// Mitsubishi GX Works2 project: ZhaoQing_ChengPinKu_Debug   PLC: Q03UDE
// 化成线2号柜

TYPE BarCylinderIO : STRUCT
  xPresentSwitch : BOOL;  (* 行程开关 *)
  xBarCylinder : BOOL;  (* 阻挡气缸 *)
  xEmpty : BOOL;  (* 为空指示 *)
  xTransportMotorCW : BOOL;  (* 输送电机正转 *)
  tLeaveDelay : TIME;  (* 放行延时 *)
  xUnload : BOOL;  (* 下料 *)
  xBarCylinderButton : BOOL;  (* 阻挡气缸 *)
  xTransportMotorCWButton : BOOL;  (* 输送电机正转按钮 *)
  xLoad : BOOL;  (* 上料 *)
  xNextRun : BOOL;  (* 下位设备开始运行 *)
  xTransportMotorCCWButton : BOOL;  (* 输送电机反转按钮 *)
  xTransportMotorCCW : BOOL;  (* 输送电机反转 *)
END_STRUCT END_TYPE

TYPE ConveyorIO : STRUCT
  xCWPresent : BOOL;  (* 正转检测有无传感器 *)
  xCCWPresent : BOOL;  (* 反转检测有无传感器 *)
  xLoad : BOOL;  (* 上料请求 *)
  xUnload : BOOL;  (* 下料请求 *)
  xMotorCW : BOOL;  (* 电机正转 *)
  xMotorCCW : BOOL;  (* 电机反转 *)
  xEmpty : BOOL;  (* 线体状态为空 *)
  xNextRun : BOOL;  (* 下段线体运行 *)
  xUnloadCCW : BOOL;  (* 下料为反转 *)
  xloadCCW : BOOL;  (* 上料为反转 *)
  xLeave : BOOL;  (* 已经离开 *)
  xForward : BOOL;  (* 正转手动 *)
  xBackward : BOOL;  (* 反转手动 *)
  xBusy : BOOL;  (* 工作中 *)
  xPutInto : BOOL;  (* 线体直接投入物料 *)
  xUnloadAlarm : BOOL;  (* 下料报警 *)
  tLoadDelay : TIME;  (* 进入延时设置 *)
  xPosLimit : BOOL;  (* 正限位 *)
  xNegLimit : BOOL;  (* 负限位 *)
  xOverWidthAlarm : BOOL;  (* 超宽报警 *)
  xLimitAlarrm : BOOL;  (* 限位报警 *)
  iDeviceID : INT;  (* 线体ID *)
END_STRUCT END_TYPE

TYPE RGVCommunication : STRUCT
  xFullLoadRequest : BOOL;  (* 满框上料请求 *)
  xFullUnloadRequest : BOOL;  (* 满框下料请求 *)
  xEmptyLoadRequest : BOOL;  (* 空框上料请求 *)
  xEmptyUnloadRequest : BOOL;  (* 空框下料请求 *)
  xFullLoadRequestAkn : BOOL;  (* 满框上料请求确认 *)
  xFullUnloadRequestAkn : BOOL;  (* 满框下料请求确认 *)
  xEmptyLoadRequestAkn : BOOL;  (* 空框上料请求确认 *)
  xEmptyUnloadRequestAkn : BOOL;  (* 空框下料请求确认 *)
  xFullLoadComplete : BOOL;  (* 满框上料完成 *)
  xFullUnloadComplete : BOOL;  (* 满框下料完成 *)
  xEmptyLoadComplete : BOOL;  (* 空框上料完成 *)
  xEmptyUnloadComplete : BOOL;  (* 空框下料完成 *)
  xFullLoadCompleteAkn : BOOL;  (* 满框上料完成确认 *)
  xFullUnloadCompleteAkn : BOOL;  (* 满框下料完成确认 *)
  xEmptyLoadCompleteAkn : BOOL;  (* 空框上料完成确认 *)
  xEmptyUnloadCompleteAkn : BOOL;  (* 空框下料完成确认 *)
END_STRUCT END_TYPE

TYPE ShuttleCarIO : STRUCT
  xReady : BOOL;  (* 准备就绪 *)
  xForward : BOOL;  (* 正转 *)
  xBackward : BOOL;  (* 反转 *)
  iCurrentPos : INT;  (* 当前位置 *)
  iDestinationPos : INT;  (* 目标位置 *)
  xCW : BOOL;  (* 正转输出 *)
  xCCW : BOOL;  (* 反转输出 *)
  xBrake : BOOL;  (* 刹车 *)
  xHomeSwitch : BOOL;  (* 零位接近开关 *)
  xPosLimit : BOOL;  (* 正限位 *)
  xNegLimit : BOOL;  (* 负限位 *)
  xMDIExe : BOOL;  (* MDI开始 *)
  xMDIDone : BOOL;  (* MDI 完成 *)
  xPassLimit : BOOL;  (* 限位屏蔽 *)
  xPosLimitCatch : BOOL;  (* 正限位捕捉 *)
  xNegLimitCatch : BOOL;  (* 负限位捕捉 *)
  xHomeExe : BOOL;  (* 开始寻零 *)
  xHomeDone : BOOL;  (* 寻零完成 *)
  xHomeBusy : BOOL;  (* 寻零中 *)
  xHomeFailed : BOOL;  (* 寻零失败 *)
  xBusy : BOOL;  (* 工作中 *)
  tArriveDelay : TIME;  (* 到位延时 *)
  xCylinder : BOOL;  (* 气缸控制 *)
  tBrakeDelay : TIME;  (* 抱闸延时 *)
  xPauseRamp : BOOL;  (* 暂停减速斜坡标志位 *)
  xPresentDetect1 : BOOL;  (* 物料有无检测1 *)
  xPresentDetect2 : BOOL;  (* 物料有无检测2 *)
  xOvertimeAlarm : BOOL;  (* 超时报警 *)
  tSetOverTime : TIME;  (* 设置超时时间 *)
  xLooseDetect : BOOL;  (* 松绳检测 *)
  xLooseAlarm : BOOL;  (* 松绳报警 *)
END_STRUCT END_TYPE

TYPE SwitchIO : STRUCT
  xLiftCylinderRetractDetect : BOOL;
  xLiftCylinderExtendDetect : BOOL;
  xLiftCylinderRetract : BOOL;
  xLiftCylinderExtend : BOOL;
  xEntryBarCylinderRetract : BOOL;
  xExitBarCylinderRetract : BOOL;
  xLiftCylinderExtendInit : BOOL;
  xEntryEnable : BOOL;
  xExitEnable : BOOL;
  xSwithEnable : BOOL;
  xLiftCylinderRetractButton : BOOL;
  xLiftCylinderExtendButton : BOOL;
  xEntryBarCylinderRetractButton : BOOL;
  xExitBarCylinderRetractButton : BOOL;
  xPutInto : BOOL;  (* 单体复位 *)
  tSetOvertime : TIME;  (* 设定超时报警时间 *)
  xOvertimeAlarm : BOOL;  (* 超时报警 *)
END_STRUCT END_TYPE

// global labels: Global1
VAR_GLOBAL
  g_xAuto AT M11 : BOOL;  (* 自动 *)
  g_xManual : BOOL;  (* 手动 *)
  g_xEStop : BOOL;  (* 急停 *)
  g_xReset : BOOL;  (* 复位 *)
  g_xStackLampRed : BOOL;
  g_xStackLampAmber : BOOL;
  g_xStackLampGreen : BOOL;
  g_xBuzzer : BOOL;
  g_xStop AT M2 : BOOL;  (* 停止 *)
  g_xLocalAutoStart AT M1 : BOOL;
  g_xRemoteAutoStart AT M0 : BOOL;
  g_xRemoteAuto AT M10 : BOOL;
  g_iState AT D40 : INT;
  g_iLocalAutoStep : INT;
  g_xError : BOOL;
  g_xStart : BOOL;  (* 启动 *)
  g_xResetSingle AT M4 : BOOL;  (* 单线体复位 *)
  g_iDeviceIDSelect AT D0 : INT;
  g_xPause AT M3 : BOOL;  (* 暂停 *)
END_VAR

// task Task_01 (event TRUE, interval 0, priority 31): Start, POU

FUNCTION_BLOCK BarCylinder
VAR_IN_OUT
  BarCylinderIO : BarCylinderIO;
END_VAR
VAR
  m_tonViaDelay : TON;  (* 卸料延时定时器 *)
  m_xViaDelay : BOOL;  (* 通过延时 *)
  m_tViaDelayElapse : TIME;  (* 通过延时当前时间 *)
  m_xInitial : BOOL;  (* 初始化 *)
END_VAR
  (***********************************************************************
阻挡器模块，
由一个行程开关，一个阻挡器，一个倍速链输送电机组成
具有手动与自动模式
xEmpty显示当前为空料的状态
xUnload为卸料信号，连接下一设备的xEmpty信号
*************************************************************************)

  (*初始化，离开延时时间设置为5秒*)
IF NOT m_xInitial THEN
	 BarCylinderIO.tLeaveDelay :=T#5s;
	m_xInitial:=1;
END_IF;
IF g_xManual THEN    (*手动*)
	BarCylinderIO.xNextRun:=0;
	IF BarCylinderIO.xBarCylinderButton THEN
		BarCylinderIO.xBarCylinder:=1;
	ELSE
		BarCylinderIO.xBarCylinder:=0;
	END_IF;
	IF BarCylinderIO.xTransportMotorCWButton 
		AND NOT BarCylinderIO.xTransportMotorCCWButton 
		AND NOT BarCylinderIO.xTransportMotorCCW   THEN
		BarCylinderIO.xTransportMotorCW:=1;
	ELSE
		BarCylinderIO.xTransportMotorCW:=0;
	END_IF;
	IF BarCylinderIO.xTransportMotorCCWButton 
		AND NOT BarCylinderIO.xTransportMotorCWButton 
		AND NOT BarCylinderIO.xTransportMotorCW   THEN
		BarCylinderIO.xTransportMotorCCW:=1;
	ELSE
		BarCylinderIO.xTransportMotorCCW:=0;
	END_IF;
END_IF;
(*离开延时定时器*)
m_tonViaDelay(IN:=NOT  BarCylinderIO.xPresentSwitch AND g_xAuto  ,PT:= BarCylinderIO.tLeaveDelay ,Q:= BarCylinderIO.xEmpty ,ET:=m_tViaDelayElapse );

IF g_xAuto THEN(*自动*)
    IF BarCylinderIO.xUnload  AND NOT BarCylinderIO.xEmpty AND NOT BarCylinderIO.xNextRun THEN(*收到卸料命令，当阻挡器不为空时*)
    	BarCylinderIO.xBarCylinder:=1;
    	BarCylinderIO.xNextRun:=1;(*确保下料命令只执行一次，防止物料在输送过程中又有卸料命令导致多事卸料*)
    	BarCylinderIO.xTransportMotorCW:=1;
    END_IF;
    IF NOT  BarCylinderIO.xUnload  THEN
    	BarCylinderIO.xNextRun:=0;
    END_IF;
    (*如果为空，气缸顶起*)
   IF  BarCylinderIO.xEmpty  THEN
   	   BarCylinderIO.xBarCylinder:=0;
   	   IF BarCylinderIO.xLoad THEN
	   	   BarCylinderIO.xTransportMotorCW:=1;
	   END_IF;
   END_IF;
   IF NOT BarCylinderIO.xUnload AND NOT  BarCylinderIO.xEmpty THEN
   	    BarCylinderIO.xTransportMotorCW:=0;
   	END_IF;
END_IF;
IF NOT g_xEStop THEN
	 BarCylinderIO.xTransportMotorCW:=0;
	 BarCylinderIO.xTransportMotorCCW:=0;
	 BarCylinderIO.xBarCylinder:=0;
END_IF;
END_FUNCTION_BLOCK

FUNCTION_BLOCK Conveyor
VAR
  tRundelay : TIME;  (* 离开延时 *)
END_VAR
VAR_IN_OUT
  ConveyorMotor : ConveyorIO;  (* 输送线输入输出 *)
END_VAR
VAR
  iStep : INT;  (* 上料步骤 *)
  m_tUnloadTimer : TIME;  (* 下料计时器 *)
  m_tonLeaveDelay : TON;  (* 离开延时定时器 *)
  m_xLeaveDelayOut : BOOL;  (* 离开延时 *)
  m_tLeaveCurrentTime : TIME;
END_VAR
VAR CONSTANT
  LOAD_UNLOAD_TIME : TIME := T#30s;  (* 延时报警常量 *)
END_VAR
VAR
  m_tonUnloadAlam : TON;  (* 下料报警定时器 *)
  m_tonLoadDelay : TON;  (* 离开延时定时器 *)
  m_xLoadDelayOut : BOOL;  (* 离开延时 *)
  m_tLoadCurrentTime : TIME;
  m_xInitial : BOOL;  (* 初始化 *)
  m_tLoadTimer : TIME;  (* 上料延时当前时间 *)
END_VAR
(*////////////////////////////////////////////////////////////////////////////////////////////////////////////
//传输线控制FB块，可控制单方向线体，双向旋转线体，支持双向上下料            
//线体初始化后为空的情况下输入xLoad信号即可进行上料动作，使用xLoadCCW信号可反方向上料
//增加了产品信息和产品种类的储存，当传输线为空和上料进行标志位为零的情况下清除产品信息和产品种类
//使用方式是在置位xLoad信号后，把产品信息和产品种类传入，等下料后自动清零
//线体不为空的情况下使用xUnload信号可进行下料动作，物料有无传感器的下降沿后出发计时器，延时断开传输线旋转
//单方向传输线体把xLoadCCW、xUnloadCCW设置为零，双向线体上料方向和下料反向的,方向固定的 把xUnloadCCW设置为1
//双方向线体双向都能上下料的要根据上料的方向来设置xLoadCCW,xUnloadCCW
//增加工作中信号xBusy当电机正转 显示为工作中
//增加上下料超时报警，xLoadAlarm，xUnloadAlarm，设定时间在LOAD_UNLOAD_TIME常量上，现在设置的为30秒
//增加xPutInto信号，用于直接投入的物料，检测开关感应到后，直接进入下料流程，上升沿有效
//离开延时改为变量 iLeaveDelay 默认为0 离开检测开关离输送线尾端比较远的线体需要根据情况设定100ms为单位
增加初始化标志位，增加进入延时时间，初始化为进入延时时间为0 ，离开延时时间为2S，通过外围接口可以更改
//修改信息  修改后请增加版本
//YAO      V1.0
///////////////////////////////////////////////////////////////////////////////////////////////////////////
********************************************************)
IF NOT m_xInitial THEN
	ConveyorMotor.tLoadDelay:=T#100ms;
	ConveyorMotor.xNegLimit:=1;
	ConveyorMotor.xPosLimit:=1;
END_IF;
m_xInitial:=1;
IF g_xAuto THEN
CASE iStep OF
	0:
	ConveyorMotor.xMotorCW:=0;
	ConveyorMotor.xMotorCCW:=0;
	ConveyorMotor.xNextRun:=0;
IF g_xEStop AND NOT ConveyorMotor.xLimitAlarrm  THEN
	IF (ConveyorMotor.xCWPresent OR ConveyorMotor.xCCWPresent)  THEN
		iStep:=3;
		ConveyorMotor.xEmpty:=0;
		ELSE
		iStep:=1;
		ConveyorMotor.xEmpty:=1;
	END_IF;
END_IF;		
	1: 
	IF ConveyorMotor.xLoad    
		AND ConveyorMotor.xMotorCW=0   
		AND ConveyorMotor.xMotorCCW=0   
		AND ConveyorMotor.xEmpty THEN	
		iStep:=2;
	END_IF;
	2: 
	IF ConveyorMotor.xloadCCW THEN
		ConveyorMotor.xMotorCCW:=1; 
		ConveyorMotor.xMotorCW:=0;
	ELSE
	    ConveyorMotor.xMotorCW:=1;  
		ConveyorMotor.xMotorCCW:=0;
	END_IF;
		m_tonLoadDelay(IN:= (ConveyorMotor.xCWPresent AND NOT ConveyorMotor.xloadCCW) 
		                                        OR (ConveyorMotor.xCCWPresent AND ConveyorMotor.xloadCCW) ,
		                               PT:= ConveyorMotor.tLoadDelay ,
		                               Q:= m_xLoadDelayOut ,
		                               ET:= m_tLoadTimer );
	    IF m_xLoadDelayOut THEN 	 
		    iStep:=3;
		END_IF;
	3:
	ConveyorMotor.xMotorCW:=0;
	ConveyorMotor.xMotorCCW:=0;
	ConveyorMotor.xEmpty:=0;
	IF ConveyorMotor.xUnload AND NOT ConveyorMotor.xOverWidthAlarm THEN 
		iStep:=4;
	END_IF;
	4:	
	IF ConveyorMotor.xUnloadCCW THEN   
		ConveyorMotor.xMotorCCW:=1;  
		ConveyorMotor.xMotorCW:=0;
		ELSE
	    ConveyorMotor.xMotorCW:=1;  
		ConveyorMotor.xMotorCCW:=0;
	END_IF;
	ConveyorMotor.xNextRun:=1; 
	IF NOT ConveyorMotor.xUnload THEN 
		istep:=0;
	END_IF;
END_CASE;
IF LDP(TRUE,ConveyorMotor.xPutInto) THEN
	iStep:=0;
END_IF;
END_IF;
IF g_xManual THEN
	iStep:=0;

	IF ConveyorMotor.xForward 
		AND ConveyorMotor.xBackward=0 
		AND ConveyorMotor.xMotorCCW=0
		AND g_xEStop THEN
		ConveyorMotor.xMotorCW:=1;
		ConveyorMotor.xMotorCCW:=0;
		ELSE
		ConveyorMotor.xMotorCW:=0;
	END_IF;

	IF ConveyorMotor.xBackward 
		AND ConveyorMotor.xForward=0 
		AND ConveyorMotor.xMotorCW=0
		AND g_xEStop  THEN
		ConveyorMotor.xMotorCCW:=1;
		conveyormotor.xMotorCW:=0;
		ELSE
		ConveyorMotor.xMotorCCW:=0;
	END_IF;
END_IF;
IF ConveyorMotor.xMotorCCW        
	OR ConveyorMotor.xMotorCW THEN  
	ConveyorMotor.xBusy:=1;
	ELSE
	ConveyorMotor.xBusy:=0;
END_IF;
m_tonUnloadAlam(IN:= iStep=4,PT:= LOAD_UNLOAD_TIME,Q:= ConveyorMotor.xUnloadAlarm,ET:= m_tUnloadTimer );
(*//复位*)
IF (*g_xReset OR*)
	 (g_xResetSingle AND ConveyorMotor.iDeviceID=g_iDeviceIDSelect)THEN (*AND ConveyorMotor.iDeviceID=g_iDeviceIDSelect  THEN*)  (* //非正常情况下切断xNextRun不会复位，通过这个标志位会出发报警*)(*增加单体复位*)
	iStep:=0;
	ConveyorMotor.xNextRun:=0; 
	ConveyorMotor.xLimitAlarrm:=0;
	ConveyorMotor.xOverWidthAlarm:=0;
END_IF;
IF iStep=3 AND (NOT ConveyorMotor.xNegLimit OR NOT ConveyorMotor.xPosLimit) THEN
	ConveyorMotor.xOverWidthAlarm:=1;
END_IF;
IF ( ((ConveyorMotor.xloadCCW AND NOT ConveyorMotor.xNegLimit)            (*反转上料，碰到负限位*)
	OR  ( NOT ConveyorMotor.xloadCCW AND NOT ConveyorMotor.xPosLimit)) (*正转上料，碰到正限位*)
    AND iStep=2) (*上料过程*)
    OR
   ( iStep=4 (*下料过程*)
	AND( (ConveyorMotor.xUnloadCCW AND NOT ConveyorMotor.xPosLimit)  
	OR (NOT ConveyorMotor.xUnloadCCW AND NOT ConveyorMotor.xNegLimit)))    
    THEN
    ConveyorMotor.xLimitAlarrm:=1;
    iStep:=0;
END_IF;
END_FUNCTION_BLOCK

PROGRAM POU
VAR
  Switch12201 : Switch;
  SwitchIO12201 : SwitchIO;
  ConveyorIO12201 : ConveyorIO;
  ConveyorIO12101 : ConveyorIO;
  Switch12202 : Switch;
  SwitchIO12202 : SwitchIO;
  ConveyorIO12102 : ConveyorIO;
  ConveyorIO12202 : ConveyorIO;
  Bar12302 : BarCylinder;
  BarIO12302 : BarCylinderIO;
  Bar12303 : BarCylinder;
  BarIO12303 : BarCylinderIO;
  Bar12304 : BarCylinder;
  BarIO12304 : BarCylinderIO;
  Bar12333 : BarCylinder;
  BarIO12333 : BarCylinderIO;
  Bar12334 : BarCylinder;
  BarIO12334 : BarCylinderIO;
  Bar12335 : BarCylinder;
  BarIO12335 : BarCylinderIO;
  Switch12203 : Switch;
  SwitchIO12203 : SwitchIO;
  ConveyorIO12203 : ConveyorIO;
  ConveyorIO12105 : ConveyorIO;
  Conveyor12106 : Conveyor;
  ConveyorIO12106 : ConveyorIO;
  Conveyor12107 : Conveyor;
  ConveyorIO12107 : ConveyorIO;
  Conveyor12108 : Conveyor;
  ConveyorIO12108 : ConveyorIO;
  Conveyor12109 : Conveyor;
  ConveyorIO12109 : ConveyorIO;
  Conveyor12110 : Conveyor;
  ConveyorIO12110 : ConveyorIO;
  Conveyor12111 : Conveyor;
  ConveyorIO12111 : ConveyorIO;
  Conveyor12112 : Conveyor;
  ConveyorIO12112 : ConveyorIO;
  Conveyor12113 : Conveyor;
  ConveyorIO12113 : ConveyorIO;
  Conveyor12114 : Conveyor;
  ConveyorIO12114 : ConveyorIO;
  Conveyor12115 : Conveyor;
  ConveyorIO12115 : ConveyorIO;
  Conveyor12116 : Conveyor;
  ConveyorIO12116 : ConveyorIO;
  Conveyor12117 : Conveyor;
  ConveyorIO12117 : ConveyorIO;
  Conveyor12118 : Conveyor;
  ConveyorIO12118 : ConveyorIO;
  Conveyor12119 : Conveyor;
  ConveyorIO12119 : ConveyorIO;
  Conveyor12120 : Conveyor;
  ConveyorIO12120 : ConveyorIO;
  Conveyor12121 : Conveyor;
  ConveyorIO12121 : ConveyorIO;
  Conveyor12122 : Conveyor;
  ConveyorIO12122 : ConveyorIO;
  Conveyor12123 : Conveyor;
  ConveyorIO12123 : ConveyorIO;
  Conveyor12124 : Conveyor;
  ConveyorIO12124 : ConveyorIO;
  Conveyor12125 : Conveyor;
  ConveyorIO12125 : ConveyorIO;
  Conveyor12126 : Conveyor;
  ConveyorIO12126 : ConveyorIO;
  Conveyor12127 : Conveyor;
  ConveyorIO12127 : ConveyorIO;
  Conveyor12128 : Conveyor;
  ConveyorIO12128 : ConveyorIO;
  Conveyor12129 : Conveyor;
  ConveyorIO12129 : ConveyorIO;
  Conveyor12130 : Conveyor;
  ConveyorIO12130 : ConveyorIO;
  Conveyor12131 : Conveyor;
  ConveyorIO12131 : ConveyorIO;
  Conveyor12132 : Conveyor;
  ConveyorIO12132 : ConveyorIO;
  Conveyor12133 : Conveyor;
  ConveyorIO12133 : ConveyorIO;
  Lifter10 : ShuttleCar;
  Lifter10IO : ShuttleCarIO;
  Lifter10IOSpeed : ShuttleCarVelocityFB;
  Conveyor10 : Conveyor;
  Conveyor10IO : ConveyorIO;
  Switch12313 : Switch;
  SwitchIO12313 : SwitchIO;
  Switch12314 : Switch;
  SwitchIO12314 : SwitchIO;
  Switch12315 : Switch;
  SwitchIO12315 : SwitchIO;
  Switch12316 : Switch;
  SwitchIO12316 : SwitchIO;
  ConveyorIO12134 : ConveyorIO;
  ConveyorIO12135 : ConveyorIO;
  ConveyorIO12136 : ConveyorIO;
  ConveyorIO12137 : ConveyorIO;
  ConveyorIO12138 : ConveyorIO;
  ConveyorIO12139 : ConveyorIO;
  ConveyorIO12140 : ConveyorIO;
  ConveyorIO12141 : ConveyorIO;
  ConveyorIO12142 : ConveyorIO;
  ConveyorIO12143 : ConveyorIO;
  ConveyorIO12144 : ConveyorIO;
  ConveyorIO12145 : ConveyorIO;
  ConveyorIO12146 : ConveyorIO;
  ConveyorIO12147 : ConveyorIO;
  ConveyorIO12148 : ConveyorIO;
  ConveyorIO12149 : ConveyorIO;
  Conveyor12139 : Conveyor;
  Conveyor12140 : Conveyor;
  Conveyor12142 : Conveyor;
  Conveyor12143 : Conveyor;
  Conveyor12148 : Conveyor;
  Conveyor12149 : Conveyor;
  m_iSwitch12313Select : INT;
  m_iSwitch12315Select : INT;
END_VAR
(*空框回流线体*)
Switch12201(ConveyorEntryIO:=ConveyorIO12101 ,
                                                        ConveyorExitIO:=ConveyorIO12201,
                                                        SwitchIO:=SwitchIO12201 );
SwitchIO12201.xLiftCylinderExtendButton:=M30;
SwitchIO12201.xLiftCylinderRetractButton:=M31;
Y203:=SwitchIO12201.xLiftCylinderExtend;
Y204:=SwitchIO12201.xLiftCylinderRetract;
SwitchIO12201.xLiftCylinderExtendDetect:=X2;
SwitchIO12201.xLiftCylinderRetractDetect:=X3;
ConveyorIO12101.xForward:=M32;
ConveyorIO12101.xCWPresent:=X1;
Y201:=ConveyorIO12101.xMotorCW;
M300:=NOT ConveyorIO12101.xEmpty;
M301:=ConveyorIO12101.xUnloadAlarm;
ConveyorIO12101.iDeviceID:=12201;
ConveyorIO12101.tLoadDelay:=T#3s;
ConveyorIO12201.xForward:=M33;
ConveyorIO12201.xCWPresent:=X4;
Y202:=ConveyorIO12201.xMotorCW;
M302:=NOT ConveyorIO12201.xEmpty;
M303:=ConveyorIO12201.xUnloadAlarm;
ConveyorIO12201.iDeviceID:=12201;

Switch12202(ConveyorEntryIO:=ConveyorIO12102 ,
                                                        ConveyorExitIO:=ConveyorIO12202,
                                                        SwitchIO:=SwitchIO12202 );
SwitchIO12202.xLiftCylinderExtendButton:=M34;
SwitchIO12202.xLiftCylinderRetractButton:=M35;
Y206:=SwitchIO12202.xLiftCylinderExtend;
Y207:=SwitchIO12202.xLiftCylinderRetract;
SwitchIO12202.xLiftCylinderExtendDetect:=X6;
SwitchIO12202.xLiftCylinderRetractDetect:=X7;
ConveyorIO12102.xForward:=M36;
ConveyorIO12102.xCWPresent:=X5;
Y205:=ConveyorIO12102.xMotorCW OR BarIO12302.xTransportMotorCW OR BarIO12335.xTransportMotorCW;
M304:=NOT ConveyorIO12102.xEmpty;
M305:=ConveyorIO12102.xUnloadAlarm;
ConveyorIO12102.iDeviceID:=12202;
ConveyorIO12102.tLoadDelay:=T#3s;
ConveyorIO12202.xForward:=M37;
ConveyorIO12202.xCWPresent:=X8;
Y208:=ConveyorIO12202.xMotorCW;
M306:=NOT ConveyorIO12202.xEmpty;
M307:=ConveyorIO12202.xUnloadAlarm;
ConveyorIO12202.iDeviceID:=12202;

Bar12302(BarCylinderIO:= BarIO12302);
BarIO12302.xBarCylinderButton:=M38;
BarIO12302.xPresentSwitch:=XB;
Y209:=BarIO12302.xBarCylinder;

Bar12303(BarCylinderIO:= BarIO12303);
BarIO12303.xBarCylinderButton:=M39;
BarIO12303.xPresentSwitch:=XE;
Y20B:=BarIO12303.xBarCylinder;

Bar12304(BarCylinderIO:= BarIO12304);
BarIO12304.xBarCylinderButton:=M40;
BarIO12304.xPresentSwitch:=XF;
Y20D:=BarIO12304.xBarCylinder;

Bar12333(BarCylinderIO:= BarIO12333);
BarIO12333.xBarCylinderButton:=M41;
BarIO12333.xPresentSwitch:=XF9;
Y2D0:=BarIO12333.xBarCylinder;
Y20C:=BarIO12333.xTransportMotorCW OR BarIO12304.xTransportMotorCW;

Bar12334(BarCylinderIO:= BarIO12334);
BarIO12334.xBarCylinderButton:=M42;
BarIO12334.xPresentSwitch:=X112;
Y2D1:=BarIO12334.xBarCylinder;
Y20A:=BarIO12334.xTransportMotorCW OR BarIO12303.xTransportMotorCW;

Bar12335(BarCylinderIO:= BarIO12335);
BarIO12335.xBarCylinderButton:=M43;
BarIO12335.xPresentSwitch:=X115;
Y2D2:=BarIO12335.xBarCylinder;
(*满框线体*)
Switch12203(ConveyorEntryIO:=ConveyorIO12203 ,
                                                        ConveyorExitIO:=ConveyorIO12105,
                                                        SwitchIO:=SwitchIO12203 );
SwitchIO12203.xLiftCylinderExtendButton:=M44;
SwitchIO12203.xLiftCylinderRetractButton:=M45;
Y210:=SwitchIO12203.xLiftCylinderExtend;
Y211:=SwitchIO12203.xLiftCylinderRetract;
SwitchIO12203.xLiftCylinderExtendDetect:=X12;
SwitchIO12203.xLiftCylinderRetractDetect:=X13;
ConveyorIO12203.xForward:=M46;
ConveyorIO12203.xCWPresent:=X14;
Y20E:=ConveyorIO12203.xMotorCW;
M308:=NOT ConveyorIO12203.xEmpty;
M309:=ConveyorIO12203.xUnloadAlarm;
ConveyorIO12203.iDeviceID:=12203;
ConveyorIO12203.tLoadDelay:=T#1s;
ConveyorIO12105.xForward:=M46;
ConveyorIO12105.xCWPresent:=X14;
Y20F:=ConveyorIO12105.xMotorCW;
M310:=NOT ConveyorIO12105.xEmpty;
M311:=ConveyorIO12105.xUnloadAlarm;
ConveyorIO12105.iDeviceID:=12203;

Conveyor12106(ConveyorMotor:=ConveyorIO12106);
ConveyorIO12106.xForward:=M47;
ConveyorIO12106.xCWPresent:=X15;
Y212:=ConveyorIO12106.xMotorCW;
M312:=NOT ConveyorIO12106.xEmpty;
M313:=ConveyorIO12106.xUnloadAlarm;
ConveyorIO12106.iDeviceID:=12106;

Conveyor12107(ConveyorMotor:=ConveyorIO12107);
ConveyorIO12107.xForward:=M48;
ConveyorIO12107.xCWPresent:=X16;
Y213:=ConveyorIO12107.xMotorCW;
M314:=NOT ConveyorIO12107.xEmpty;
M315:=ConveyorIO12107.xUnloadAlarm;
ConveyorIO12107.iDeviceID:=12107;

Conveyor12108(ConveyorMotor:=ConveyorIO12108);
ConveyorIO12108.xForward:=M49;
ConveyorIO12108.xCWPresent:=X17;
Y214:=ConveyorIO12108.xMotorCW;
M316:=NOT ConveyorIO12108.xEmpty;
M317:=ConveyorIO12108.xUnloadAlarm;
ConveyorIO12108.iDeviceID:=12108;

Conveyor12109(ConveyorMotor:=ConveyorIO12109);
ConveyorIO12109.xForward:=M50;
ConveyorIO12109.xCWPresent:=X18;
Y215:=ConveyorIO12109.xMotorCW;
M318:=NOT ConveyorIO12109.xEmpty;
M319:=ConveyorIO12109.xUnloadAlarm;
ConveyorIO12109.iDeviceID:=12109;

Conveyor12110(ConveyorMotor:=ConveyorIO12110);
ConveyorIO12110.xForward:=M51;
ConveyorIO12110.xCWPresent:=X19;
Y216:=ConveyorIO12110.xMotorCW;
M320:=NOT ConveyorIO12110.xEmpty;
M321:=ConveyorIO12110.xUnloadAlarm;
ConveyorIO12110.iDeviceID:=12110;

Conveyor12111(ConveyorMotor:=ConveyorIO12111);
ConveyorIO12111.xForward:=M52;
ConveyorIO12111.xCWPresent:=X1A;
Y217:=ConveyorIO12111.xMotorCW;
M322:=NOT ConveyorIO12111.xEmpty;
M323:=ConveyorIO12111.xUnloadAlarm;
ConveyorIO12111.iDeviceID:=12111;

Conveyor12112(ConveyorMotor:=ConveyorIO12112);
ConveyorIO12112.xForward:=M53;
ConveyorIO12112.xCWPresent:=X1B;
Y218:=ConveyorIO12112.xMotorCW;
M324:=NOT ConveyorIO12112.xEmpty;
M325:=ConveyorIO12112.xUnloadAlarm;
ConveyorIO12112.iDeviceID:=12112;

Conveyor12113(ConveyorMotor:=ConveyorIO12113);
ConveyorIO12113.xForward:=M54;
ConveyorIO12113.xCWPresent:=X1C;
Y219:=ConveyorIO12113.xMotorCW;
M326:=NOT ConveyorIO12113.xEmpty;
M327:=ConveyorIO12113.xUnloadAlarm;
ConveyorIO12113.iDeviceID:=12113;

Conveyor12114(ConveyorMotor:=ConveyorIO12114);
ConveyorIO12114.xForward:=M55;
ConveyorIO12114.xCWPresent:=X1D;
Y21A:=ConveyorIO12114.xMotorCW;
M328:=NOT ConveyorIO12114.xEmpty;
M329:=ConveyorIO12114.xUnloadAlarm;
ConveyorIO12114.iDeviceID:=12114;

Conveyor12115(ConveyorMotor:=ConveyorIO12115);
ConveyorIO12115.xForward:=M56;
ConveyorIO12115.xCWPresent:=X1E;
Y21B:=ConveyorIO12115.xMotorCW;
M330:=NOT ConveyorIO12115.xEmpty;
M331:=ConveyorIO12115.xUnloadAlarm;
ConveyorIO12115.iDeviceID:=12115;

Conveyor12116(ConveyorMotor:=ConveyorIO12116);
ConveyorIO12116.xForward:=M57;
ConveyorIO12116.xCWPresent:=X1F;
Y21C:=ConveyorIO12116.xMotorCW;
M332:=NOT ConveyorIO12116.xEmpty;
M333:=ConveyorIO12116.xUnloadAlarm;
ConveyorIO12116.iDeviceID:=12116;

Conveyor12117(ConveyorMotor:=ConveyorIO12117);
ConveyorIO12117.xForward:=M58;
ConveyorIO12117.xCWPresent:=X20;
Y21D:=ConveyorIO12117.xMotorCW;
M334:=NOT ConveyorIO12117.xEmpty;
M335:=ConveyorIO12117.xUnloadAlarm;
ConveyorIO12117.iDeviceID:=12117;

Conveyor12118(ConveyorMotor:=ConveyorIO12118);
ConveyorIO12118.xForward:=M59;
ConveyorIO12118.xCWPresent:=X21;
Y21E:=ConveyorIO12118.xMotorCW;
M336:=NOT ConveyorIO12118.xEmpty;
M337:=ConveyorIO12118.xUnloadAlarm;
ConveyorIO12118.iDeviceID:=12118;

Conveyor12119(ConveyorMotor:=ConveyorIO12119);
ConveyorIO12119.xForward:=M60;
ConveyorIO12119.xCWPresent:=X22;
Y21F:=ConveyorIO12119.xMotorCW;
M338:=NOT ConveyorIO12119.xEmpty;
M339:=ConveyorIO12119.xUnloadAlarm;
ConveyorIO12119.iDeviceID:=12119;

Conveyor12120(ConveyorMotor:=ConveyorIO12120);
ConveyorIO12120.xForward:=M61;
ConveyorIO12120.xCWPresent:=X23;
Y220:=ConveyorIO12120.xMotorCW;
M340:=NOT ConveyorIO12120.xEmpty;
M341:=ConveyorIO12120.xUnloadAlarm;
ConveyorIO12120.iDeviceID:=12120;

Conveyor12121(ConveyorMotor:=ConveyorIO12121);
ConveyorIO12121.xForward:=M62;
ConveyorIO12121.xCWPresent:=X24;
Y221:=ConveyorIO12121.xMotorCW;
M342:=NOT ConveyorIO12121.xEmpty;
M343:=ConveyorIO12121.xUnloadAlarm;
ConveyorIO12121.iDeviceID:=12121;

Conveyor12122(ConveyorMotor:=ConveyorIO12122);
ConveyorIO12122.xForward:=M63;
ConveyorIO12122.xCWPresent:=X25;
Y222:=ConveyorIO12122.xMotorCW;
M344:=NOT ConveyorIO12122.xEmpty;
M345:=ConveyorIO12122.xUnloadAlarm;
ConveyorIO12122.iDeviceID:=12122;

Conveyor12123(ConveyorMotor:=ConveyorIO12123);
ConveyorIO12123.xForward:=M64;
ConveyorIO12123.xCWPresent:=X26;
Y223:=ConveyorIO12123.xMotorCW;
M346:=NOT ConveyorIO12123.xEmpty;
M347:=ConveyorIO12123.xUnloadAlarm;
ConveyorIO12123.iDeviceID:=12123;

Conveyor12124(ConveyorMotor:=ConveyorIO12124);
ConveyorIO12124.xForward:=M65;
ConveyorIO12124.xCWPresent:=X27;
Y224:=ConveyorIO12124.xMotorCW;
M348:=NOT ConveyorIO12124.xEmpty;
M349:=ConveyorIO12124.xUnloadAlarm;
ConveyorIO12124.iDeviceID:=12124;

Conveyor12125(ConveyorMotor:=ConveyorIO12125);
ConveyorIO12125.xForward:=M66;
ConveyorIO12125.xCWPresent:=X28;
Y225:=ConveyorIO12125.xMotorCW;
M350:=NOT ConveyorIO12125.xEmpty;
M351:=ConveyorIO12125.xUnloadAlarm;
ConveyorIO12125.iDeviceID:=12125;

Conveyor12126(ConveyorMotor:=ConveyorIO12126);
ConveyorIO12126.xForward:=M67;
ConveyorIO12126.xCWPresent:=X29;
Y226:=ConveyorIO12126.xMotorCW;
M352:=NOT ConveyorIO12126.xEmpty;
M353:=ConveyorIO12126.xUnloadAlarm;
ConveyorIO12126.iDeviceID:=12126;

Conveyor12127(ConveyorMotor:=ConveyorIO12127);
ConveyorIO12127.xForward:=M68;
ConveyorIO12127.xCWPresent:=X2A;
Y227:=ConveyorIO12127.xMotorCW;
M354:=NOT ConveyorIO12127.xEmpty;
M355:=ConveyorIO12127.xUnloadAlarm;
ConveyorIO12127.iDeviceID:=12127;

Conveyor12128(ConveyorMotor:=ConveyorIO12128);
ConveyorIO12128.xForward:=M69;
ConveyorIO12128.xCWPresent:=X2B;
Y228:=ConveyorIO12128.xMotorCW;
M356:=NOT ConveyorIO12128.xEmpty;
M357:=ConveyorIO12128.xUnloadAlarm;
ConveyorIO12128.iDeviceID:=12128;

Conveyor12129(ConveyorMotor:=ConveyorIO12129);
ConveyorIO12129.xForward:=M70;
ConveyorIO12129.xCWPresent:=X2C;
Y229:=ConveyorIO12129.xMotorCW;
M358:=NOT ConveyorIO12129.xEmpty;
M359:=ConveyorIO12129.xUnloadAlarm;
ConveyorIO12129.iDeviceID:=12129;

Conveyor12130(ConveyorMotor:=ConveyorIO12130);
ConveyorIO12130.xForward:=M71;
ConveyorIO12130.xCWPresent:=X2D;
Y22A:=ConveyorIO12130.xMotorCW;
M360:=NOT ConveyorIO12130.xEmpty;
M361:=ConveyorIO12130.xUnloadAlarm;
ConveyorIO12130.iDeviceID:=12130;

Conveyor12131(ConveyorMotor:=ConveyorIO12131);
ConveyorIO12131.xForward:=M72;
ConveyorIO12131.xCWPresent:=X2E;
Y22B:=ConveyorIO12131.xMotorCW;
M362:=NOT ConveyorIO12131.xEmpty;
M363:=ConveyorIO12131.xUnloadAlarm;
ConveyorIO12131.iDeviceID:=12131;

Conveyor12132(ConveyorMotor:=ConveyorIO12132);
ConveyorIO12132.xForward:=M73;
ConveyorIO12132.xCWPresent:=X2F;
Y22C:=ConveyorIO12132.xMotorCW;
M364:=NOT ConveyorIO12132.xEmpty;
M365:=ConveyorIO12132.xUnloadAlarm;
ConveyorIO12132.iDeviceID:=12132;

Conveyor12133(ConveyorMotor:=ConveyorIO12133);
ConveyorIO12133.xForward:=M74;
ConveyorIO12133.xCWPresent:=X30;
Y22D:=ConveyorIO12133.xMotorCW;
M366:=NOT ConveyorIO12133.xEmpty;
M367:=ConveyorIO12133.xUnloadAlarm;
ConveyorIO12133.iDeviceID:=12133;

(*提升机10*)
Lifter10(ShuttleCarInOut:=Lifter10IO);
ShuttleCarCurrentPosition(XC1 OR XC2 OR XC3 ,XC1 ,XC2, XC3, Lifter10IO.iCurrentPos);
Lifter10IOSpeed(xEnable:= g_xAuto,
                        xMotorCW:=Lifter10IO.xCW ,
                        xMotorCCW:= Lifter10IO.xCCW,
                        xPosition1Switch:= XC1,
                        xDecelerationSwitch:= XC0 ,
	                    xPosition2Switch:= XC3 ,
	                   xHighSpeed:= Y292 );
Lifter10IO.xReady:=XBA;
Lifter10IO.xLooseDetect:=XC6;
Lifter10IO.xForward:=M75 OR XC7;
Lifter10IO.xBackward:=M76 OR XC8;
Lifter10IO.xPosLimit:=XC4;
Lifter10IO.xNegLimit:=XC5;
Y290:=Lifter10IO.xCW;
Y291:=Lifter10IO.xCCW;
Y295:=Lifter10IO.xBrake;
Lifter10IO.tArriveDelay:=T#500ms;

Conveyor10(ConveyorMotor:=Conveyor10IO);
Conveyor10IO.xForward:=M77;
Conveyor10IO.xBackward:=M78;
Conveyor10IO.xCWPresent:=XC9;
Conveyor10IO.xCCWPresent:=XCA;
Y296:=Conveyor10IO.xMotorCW;
Y297:=Conveyor10IO.xMotorCCW;
M368:=NOT Conveyor10IO.xEmpty;
M369:=Conveyor10IO.xUnloadAlarm;
Conveyor10IO.iDeviceID:=10;

(*1巷道入库线体*)
Switch12313(ConveyorEntryIO:=ConveyorIO12134 ,
                                                        ConveyorExitIO:=ConveyorIO12138 ,
                                                        SwitchIO:=SwitchIO12313);
SwitchIO12313.xLiftCylinderExtendButton:=M79;
SwitchIO12313.xLiftCylinderRetractButton:=M80;
SwitchIO12313.xExitBarCylinderRetractButton:=M81;
Y233:=SwitchIO12313.xExitBarCylinderRetract OR m_iSwitch12313Select=2 ;
Y234:=SwitchIO12313.xExitBarCylinderRetract ;
Y240:=SwitchIO12313.xLiftCylinderExtend;
Y241:=SwitchIO12313.xLiftCylinderRetract;
SwitchIO12313.xLiftCylinderExtendDetect:=X4A;
SwitchIO12313.xLiftCylinderRetractDetect:=X4B;
ConveyorIO12134.xForward:=M81;
ConveyorIO12134.xCWPresent:=((m_iSwitch12313Select=1 OR m_iSwitch12313Select=0) AND   X36) OR (m_iSwitch12313Select=2 AND X39);
Y22E:=ConveyorIO12134.xMotorCW;
ConveyorIO12134.tLoadDelay:=T#3s;
M370:=NOT ConveyorIO12134.xEmpty;
M371:=ConveyorIO12134.xUnloadAlarm;
ConveyorIO12134.iDeviceID:=12313;
ConveyorIO12138.xForward:=M82;
ConveyorIO12138.xCWPresent:=((m_iSwitch12313Select=1 OR m_iSwitch12313Select=0) AND   X36) OR (m_iSwitch12313Select=2 AND X39);
Y249:=ConveyorIO12138.xMotorCW;
M372:=NOT ConveyorIO12138.xEmpty;
M373:=ConveyorIO12138.xUnloadAlarm;
ConveyorIO12138.iDeviceID:=12313;

(*1巷道出库线体*)
Switch12314(ConveyorEntryIO:=ConveyorIO12141 ,
                                                        ConveyorExitIO:=ConveyorIO12135 ,
                                                        SwitchIO:=SwitchIO12314 );
SwitchIO12314 .xLiftCylinderExtendButton:=M83;
SwitchIO12314 .xLiftCylinderRetractButton:=M84;
Y242:=SwitchIO12314 .xLiftCylinderExtend;
Y243:=SwitchIO12314 .xLiftCylinderRetract;
SwitchIO12314 .xLiftCylinderExtendDetect:=X4C;
SwitchIO12314 .xLiftCylinderRetractDetect:=X4D;
ConveyorIO12141.xForward:=M85;
ConveyorIO12141.xCWPresent:=X3D OR X3E;
Y24C:=ConveyorIO12141.xMotorCW;
ConveyorIO12141.tLoadDelay:=T#2s;
M374:=NOT ConveyorIO12141.xEmpty;
M375:=ConveyorIO12141.xUnloadAlarm;
ConveyorIO12141.iDeviceID:=12314;
ConveyorIO12135.xForward:=M46;
ConveyorIO12135.xCWPresent:=X3D OR X3E;
Y22F:=ConveyorIO12135.xMotorCW;
M376:=NOT ConveyorIO12135.xEmpty;
M377:=ConveyorIO12135.xUnloadAlarm;
ConveyorIO12135.iDeviceID:=12314;

(*2巷道入库线体*)
Switch12315(ConveyorEntryIO:=ConveyorIO12136 ,
                                                        ConveyorExitIO:=ConveyorIO12144 ,
                                                        SwitchIO:=SwitchIO12315);
SwitchIO12315.xLiftCylinderExtendButton:=M79;
SwitchIO12315.xLiftCylinderRetractButton:=M80;
SwitchIO12315.xExitBarCylinderRetractButton:=M81;
Y237:=SwitchIO12315.xExitBarCylinderRetract OR m_iSwitch12315Select=2 ;
Y238:=SwitchIO12315.xExitBarCylinderRetract ;
Y244:=SwitchIO12315.xLiftCylinderExtend;
Y245:=SwitchIO12315.xLiftCylinderRetract;
SwitchIO12315.xLiftCylinderExtendDetect:=X4A;
SwitchIO12315.xLiftCylinderRetractDetect:=X4B;
ConveyorIO12136 .xForward:=M82;
ConveyorIO12136 .xCWPresent:=((m_iSwitch12315Select=1 OR m_iSwitch12315Select=0) AND   X44) OR (m_iSwitch12315Select=2 AND X47);
Y230:=ConveyorIO12136 .xMotorCW;
ConveyorIO12136 .tLoadDelay:=T#3s;
M378:=NOT ConveyorIO12136 .xEmpty;
M379:=ConveyorIO12136 .xUnloadAlarm;
ConveyorIO12136 .iDeviceID:=12315;
ConveyorIO12144.xForward:=M83;
ConveyorIO12144.xCWPresent:=((m_iSwitch12315Select=1 OR m_iSwitch12315Select=0) AND   X44) OR (m_iSwitch12315Select=2 AND X47);
Y24F:=ConveyorIO12144.xMotorCW;
M380:=NOT ConveyorIO12144.xEmpty;
M381:=ConveyorIO12144.xUnloadAlarm;
ConveyorIO12144.iDeviceID:=12315;

(*2巷道出库线体*)
Switch12316(ConveyorEntryIO:=ConveyorIO12147 ,
                                                        ConveyorExitIO:=ConveyorIO12137 ,
                                                        SwitchIO:=SwitchIO12316 );
SwitchIO12316 .xLiftCylinderExtendButton:=M84;
SwitchIO12316 .xLiftCylinderRetractButton:=M85;
Y242:=SwitchIO12316 .xLiftCylinderExtend;
Y243:=SwitchIO12316 .xLiftCylinderRetract;
SwitchIO12316 .xLiftCylinderExtendDetect:=X4C;
SwitchIO12316 .xLiftCylinderRetractDetect:=X4D;
ConveyorIO12147.xForward:=M86;
ConveyorIO12147.xCWPresent:=X3D OR X3E;
Y24C:=ConveyorIO12147.xMotorCW;
ConveyorIO12147.tLoadDelay:=T#2s;
M374:=NOT ConveyorIO12147.xEmpty;
M375:=ConveyorIO12147.xUnloadAlarm;
ConveyorIO12147.iDeviceID:=12316;
ConveyorIO12137.xForward:=M87;
ConveyorIO12137.xCWPresent:=X3D OR X3E;
Y22F:=ConveyorIO12137.xMotorCW;
M376:=NOT ConveyorIO12137.xEmpty;
M377:=ConveyorIO12137.xUnloadAlarm;
ConveyorIO12137.iDeviceID:=12316;
END_PROGRAM

FUNCTION_BLOCK ShuttleCar
VAR_IN_OUT
  ShuttleCarInOut : ShuttleCarIO;
END_VAR
VAR
  m_tonBrakeDelay : TON;  (* 延时 *)
  m_tBrakeDelayCurrentTime : TIME;
  m_tonArriveDelay : TON;  (* 到达延时计时器 *)
  m_xArriveDelay : BOOL;  (* 到达延时 *)
  m_tArriveDelayCurrentTime : TIME;  (* 到达延时当前时间 *)
  m_xInit : BOOL;  (* 初始化标志位 *)
  m_tonPauseDelay : TON;  (* 暂停减速 *)
  m_tPauseDelayCurrentTime : TIME;  (* 暂停延时当前时间 *)
  m_tonOvertimeAlarm : TON;  (* 超时报警定时器 *)
  m_tOvertimeCurrentTime : TIME;  (* 超时报警当前时间 *)
END_VAR
(*******************************************************************
输送小车程序，可用于使用认址片控制位置的输送车程序，可用于控制提升机，
使用了限位捕捉程序防止小车惯性过大冲过限位后继续行走，捕捉程序采用反
转复位，这样设计有弊端可能反转复位后车的位置并没有回到限位以内,当两个
限位同时碰到的时候，会使运料小车进入死锁状态，通过xPassLimit来解开死锁，
可以在触摸屏中使用一个带权限的按钮来进行控制，配合ShuttleCarCurrentPos
函数来计算位置信息
增加自动开始后将当前位置置为零的信号防止设备停在两个位置开关的中间
修改信息  修改后请增加版本
2018-1-22增加到位延时：到位延时时间可以设置，适应双向到位的位置开关，通过调整延时时间让穿梭车停在到位开关的中间
增加气缸控制信号
增加抱闸延时
增加超时报警
YAO      V1.0
2018-1-22 YAO V1.1
********************************************************************)
IF NOT m_xInit THEN
	ShuttleCarInOut.tArriveDelay:=T#0s;   (*到位延时初始化为0*)
	ShuttleCarInOut.tBrakeDelay:=T#100ms;(*抱闸延时初始化为100ms*)
	ShuttleCarInOut.tSetOverTime:=T#60s;(*超时报警初始化为1分钟*)
	m_xInit:=1;
END_IF;
(*如果是气缸的话屏蔽限位和Ready信号*)
IF ShuttleCarInOut.xCylinder THEN
	ShuttleCarInOut.xPosLimit:=1;
	ShuttleCarInOut.xNegLimit:=1;
	ShuttleCarInOut.xReady:=1;
END_IF;
(*限位捕捉，防止冲过限位开关，反转后复位*)
ShuttleCarInOut.xPosLimitCatch:=LDF(TRUE,ShuttleCarInOut.xPosLimit) OR ShuttleCarInOut.xPosLimitCatch;
IF ShuttleCarInOut.xCCW THEN  
	ShuttleCarInOut.xPosLimitCatch:=0;
END_IF;

ShuttleCarInOut.xNegLimitCatch:=LDF(TRUE,ShuttleCarInOut.xNegLimit) OR ShuttleCarInOut.xNegLimitCatch;
(*松绳报警*)
IF LDP(TRUE,ShuttleCarInOut.xLooseDetect) THEN	
	ShuttleCarInOut.xLooseAlarm:=1;
END_IF;
(*提升复位报警*)
IF ShuttleCarInOut.xCW AND NOT  ShuttleCarInOut.xLooseDetect THEN   
	ShuttleCarInOut.xLooseAlarm:=0; 
END_IF;

IF ShuttleCarInOut.xCW THEN   
	ShuttleCarInOut.xNegLimitCatch:=0; 
END_IF;

IF ShuttleCarInOut.xPassLimit OR
	g_xReset OR   (*增加复位按钮*)
	(ShuttleCarInOut.xNegLimitCatch 
	AND ShuttleCarInOut.xPosLimitCatch)  THEN  
	ShuttleCarInOut.xNegLimitCatch:=0; 
	ShuttleCarInOut.xPosLimitCatch:=0;
	ShuttleCarInOut.xLooseAlarm:=0;
END_IF;
IF ShuttleCarInOut.xReady AND g_xEStop THEN
(*手动*)
    IF g_xManual THEN  
	    IF ShuttleCarInOut.xForward 
			AND ShuttleCarInOut.xBackward=0 
			AND ShuttleCarInOut.xCCW=0 
			AND ShuttleCarInOut.xPosLimitCatch=0  THEN
		    ShuttleCarInOut.xCW:=1;
		    ELSE
		    ShuttleCarInOut.xCW:=0;
	    END_IF;
	    IF ShuttleCarInOut.xBackward 
			AND ShuttleCarInOut.xForward=0 
			AND ShuttleCarInOut.xCW=0 
			AND ShuttleCarInOut.xNegLimitCatch=0 
			AND ShuttleCarInOut.xLooseAlarm=0
			AND G_xEStop THEN  
		    ShuttleCarInOut.xCCW:=1;
		    ELSE
		    ShuttleCarInOut.xCCW:=0;
	    END_IF;
    END_IF;
    (**********)
(*自动*)
  IF g_xAuto  THEN  
  	(*点动*)
 		IF LDP(TRUE,ShuttleCarInOut.xForward) THEN
 			ShuttleCarInOut.xMDIExe:=1;
			ShuttleCarInOut.iDestinationPos:=ShuttleCarInOut.iCurrentPos+1;
		END_IF;
		IF LDP(TRUE,ShuttleCarInOut.xBackward) THEN
			ShuttleCarInOut.xMDIExe:=1;
			ShuttleCarInOut.iDestinationPos:=ShuttleCarInOut.iCurrentPos-1;
		END_IF;	 
	(*>>>>>>>>>>>>>>>>>>>>>>>>>>>>>>>>>>>>>*)	
	  IF ShuttleCarInOut.xMDIExe AND ShuttleCarInOut.iDestinationPos<>0 THEN	
	    IF ShuttleCarInOut.iCurrentPos<ShuttleCarInOut.iDestinationPos AND ShuttleCarInOut.xPosLimitCatch=0 THEN   (*正转*)
			ShuttleCarInOut.xCW:=1;
			ShuttleCarInOut.xCCW:=0;
			ShuttleCarInOut.xMDIDone:=0;
		END_IF;

		IF ShuttleCarInOut.iCurrentPos>ShuttleCarInOut.iDestinationPos AND ShuttleCarInOut.xNegLimitCatch=0 AND ShuttleCarInOut.xLooseAlarm=0 THEN   (*反转*)
			ShuttleCarInOut.xCCW:=1;
			ShuttleCarInOut.xCW:=0;
			ShuttleCarInOut.xMDIDone:=0;
		END_IF;
	m_tonArriveDelay(IN:= ShuttleCarInOut.iCurrentPos=ShuttleCarInOut.iDestinationPos ,
	                                    PT:= ShuttleCarInOut.tArriveDelay ,
	                                    Q:= m_xArriveDelay ,
	                                    ET:= m_tArriveDelayCurrentTime);
	     (*到位延时时间可以设置，适应双向到位的位置开关，通过调整延时时间让穿梭车停在到位开关的中间*)
		IF m_xArriveDelay AND NOT ShuttleCarInOut.xCylinder THEN
			ShuttleCarInOut.xCW:=0;
			ShuttleCarInOut.xCCW:=0;
			ShuttleCarInOut.xMDIDone:=1;
			ELSE
			ShuttleCarInOut.xMDIDone:=0;
		END_IF;

		IF ShuttleCarInOut.xPosLimitCatch THEN
			ShuttleCarInOut.xCW:=0;
			ShuttleCarInOut.xMDIDone:=0;
		END_IF;

		IF ShuttleCarInOut.xNegLimitCatch THEN
			ShuttleCarInOut.xCCW:=0;
			ShuttleCarInOut.xMDIDone:=0;
		END_IF;
		ELSE
		ShuttleCarInOut.xCW:=0;
		ShuttleCarInOut.xCCW:=0;
		ShuttleCarInOut.xMDIDone:=0;
	  END_IF;
	END_IF;
	ELSE  (*无就绪信号   或急停的情况下*)
		ShuttleCarInOut.xCW:=0;
		ShuttleCarInOut.xCCW:=0;	
END_IF;
    (*抱闸延时*)
m_tonBrakeDelay(IN:= ShuttleCarInOut.xCW OR ShuttleCarInOut.xCCW,
                                    PT:= ShuttleCarInOut.tBrakeDelay,
                                    Q:=ShuttleCarInOut.xBrake ,
                                    ET:= m_tBrakeDelayCurrentTime);

(*自动上电后把当前位置清零，防止穿梭车不在开关位置*)
IF LDP(TRUE,g_xAuto) THEN
	ShuttleCarInOut.iCurrentPos:=0;
END_IF;
IF ShuttleCarInOut.xCW OR ShuttleCarInOut.xCCW THEN
	ShuttleCarInOut.xBusy:=1;
	ELSE
	ShuttleCarInout.xBusy:=0;
END_IF;

(*暂停，带延时减速斜坡，ShuttleCarInOut.xPauseRamp为减速斜坡输出位*)
m_tonPauseDelay(IN:=g_xPause,PT:= T#2s ,Q:=ShuttleCarInOut.xPauseRamp,ET:= m_tPauseDelayCurrentTime );
IF ShuttleCarInOut.xPauseRamp THEN
	ShuttleCarInOut.xCW:=0;
	ShuttleCarInOut.xCCW:=0;
	ShuttleCarInOut.xBrake:=0;
END_IF;
(*超时报警*)
m_tonOvertimeAlarm(IN:= ShuttleCarInOut.xMDIExe AND (ShuttleCarInOut.iCurrentPos<>ShuttleCarInOut.iDestinationPos) ,
                                           PT:= ShuttleCarInOut.tSetOverTime,
                                           Q:= ShuttleCarInOut.xOvertimeAlarm ,
                                           ET:= m_tOvertimeCurrentTime );
END_FUNCTION_BLOCK

FUNCTION ShuttleCarCurrentPosition
VAR_INPUT
  xPosition1 : BOOL;
  xPosition2 : BOOL;
  xPosition3 : BOOL;
END_VAR
(************************************
计算输送车当前位置的函数
**************************************)
IF xPosition1 THEN
	ShuttleCarCurrentPosition:=1;
END_IF;
IF xPosition2 THEN
	ShuttleCarCurrentPosition:=2;
END_IF;
IF xPosition3 THEN
	ShuttleCarCurrentPosition:=3;
END_IF;
END_FUNCTION

FUNCTION_BLOCK ShuttleCarVelocityFB
VAR_INPUT
  xEnable : BOOL;  (* 使能 *)
  xMotorCW : BOOL;  (* 电机正转 *)
  xMotorCCW : BOOL;  (* 电机反转 *)
  xPosition1Switch : BOOL;  (* 位置1开关 *)
  xDecelerationSwitch : BOOL;  (* 减速开关 *)
  xPosition2Switch : BOOL;  (* 位置2开关 *)
END_VAR
VAR
  iFloor : INT;  (* 层数 *)
END_VAR
VAR_OUTPUT
  xHighSpeed : BOOL;
END_VAR
IF xEnable THEN
	(*电机旋转，并且在位置开关上的时候触发加速*)
	IF( LDP(TRUE,xMotorCW) AND xPosition1Switch ) OR (  LDP(TRUE,xMotorCCW) AND xPosition2Switch) THEN
		xHighSpeed:=1;
		iFloor:=0;
	END_IF;
	IF LDF(TRUE,xMotorCW) OR LDF(TRUE,xMotorCCW) THEN
		xHighSpeed:=0;
    END_IF;
	IF LDP(TRUE,xDecelerationSwitch) THEN
		iFloor:=iFloor+1;
	END_IF;
	IF iFloor=2 THEN
		xHighSpeed:=0;
		iFloor:=0;
	END_IF;
ELSE
    xHighSpeed:=0;
END_IF;
END_FUNCTION_BLOCK

PROGRAM Start
IF g_xReset THEN
	SM50:=1;
ELSE
	SM50:=0;
END_IF;
CASE g_iState OF
	0: 
		g_xManual:=1;
		g_xAuto:=0;	
		g_xStackLampAmber:=1;
		g_xStackLampGreen:=0;
		g_xRemoteAuto:=0;
	1:
		g_xManual:=0;
		g_xAuto:=1;
		g_xStackLampGreen:=1;
		g_xStackLampAmber:=0;
		g_xRemoteAuto:=0;
	2:	
        g_xRemoteAuto:=1;
        g_xStackLampGreen:=1;
        g_xStackLampAmber:=0;
        g_xAuto:=0;
		g_xManual:=0;
END_CASE;
IF g_xLocalAutoStart THEN  
	g_iState:=1;
END_IF;

IF g_xStop OR g_xEStop=0 THEN 
	g_iState:=0;
END_IF;
IF g_xRemoteAutoStart THEN
	g_iState:=2;
END_IF;
END_PROGRAM

FUNCTION_BLOCK Switch
VAR_IN_OUT
  ConveyorEntryIO : ConveyorIO;
  ConveyorExitIO : ConveyorIO;
  SwitchIO : SwitchIO;
END_VAR
VAR
  ConveyorEntry : Conveyor;
  ConveyorExit : Conveyor;
  iStep : INT;
  m_tonLiftCylinderDelay : TON;  (* 顶升延时 *)
  m_xLiftCylinderDelay : BOOL;
  m_tLiftCylinderDelay : TIME;
  m_tonExitBarDelay : TON;  (* 退出阻挡器延时 *)
  m_tExitBarDelay : TIME;
  m_xExitBarDelay : BOOL;
  m_xInitial : BOOL;
  m_tonCylinderOvertime : TON;  (* 气缸超时报警定时器 *)
  m_tCylinderOvertimeCurrent : TIME;
END_VAR
(**************************************************
顶升移载模块，抽象为一条输入输线 ，一条输出输送线
一个进入阻挡器，一个放出阻挡器，和一个顶升气缸的控制
程序思路比较混乱，接口不清晰，需要整改
直接放行的时候有问题
switchEnable =0的时候   离开线体的PutInto有问题
增加xPutInto程序
12-17日   V1.0
***************************************************)
ConveyorEntry(ConveyorMotor:=ConveyorEntryIO);
ConveyorExit(ConveyorMotor:=ConveyorExitIO);


IF NOT m_xInitial THEN
	
	m_xInitial:=1;
END_IF;
IF g_xAuto THEN
	CASE iStep OF
		0:(*初始化*)
		ConveyorEntryIO.xLoad:=0;
		ConveyorEntryIO.xUnload:=0;
		ConveyorEntryIO.xPutInto:=0;
		ConveyorExitIO.xLoad:=0;
		ConveyorExitIo.xUnload:=0;
		ConveyorExitIO.xPutInto:=0;
		SwitchIO.xEntryBarCylinderRetract:=0;
		SwitchIO.xExitBarCylinderRetract:=0;
		IF SwitchIO.xLiftCylinderExtendInit THEN
			SwitchIO.xLiftCylinderExtend:=1;
			SwitchIO.xLiftCylinderRetract:=0;
		    IF SwitchIO.xLiftCylinderExtendDetect THEN
			    iStep:=1;
		     END_IF; 
		ELSE
			SwitchIO.xLiftCylinderExtend:=0;
			SwitchIO.xLiftCylinderRetract:=1;	
		    IF SwitchIO.xLiftCylinderRetractDetect THEN
			    iStep:=1;
		    END_IF;		
		END_IF;
		1:(*上料*)
        IF SwitchIO.xEntryEnable AND ConveyorEntryIO.xEmpty AND ConveyorExitIO.xEmpty THEN
        	SwitchIO.xEntryBarCylinderRetract:=1;
        	ConveyorEntryIO.xLoad:=1;
        END_IF;
        IF ConveyorEntryIO.xEmpty=0 THEN
        	SwitchIO.xEntryBarCylinderRetract:=0;
        	ConveyorEntryIO.xLoad:=0;
        	ConveyorExitIO.xPutInto:=1;
        END_IF;
        IF m_xLiftCylinderDelay AND  SwitchIO.xSwithEnable THEN
        	 iStep:=2;
        END_IF;
        IF SwitchIO.xSwithEnable=0 AND m_xLiftCylinderDelay  THEN
        	 iStep:=3;
        END_IF;
		2:(*顶升*)
			SwitchIO.xExitBarCylinderRetract:=0;
		    IF SwitchIO.xLiftCylinderExtendInit THEN
			    SwitchIO.xLiftCylinderExtend:=0;
			    SwitchIO.xLiftCylinderRetract:=1;
		    ELSE
			    SwitchIO.xLiftCylinderExtend:=1;
			    SwitchIO.xLiftCylinderRetract:=0;			
		   END_IF;

		  IF SwitchIO.xLiftCylinderExtendInit THEN
		  	IF SwitchIO.xLiftCylinderRetractDetect THEN
		  		iStep:=4;
		  	END_IF;
		  	ELSE
		  	IF SwitchIO.xLiftCylinderExtendDetect THEN
		      iStep:=4; 
		  	END_IF;
		  END_IF;
		  3:(*放行*)	
		  	SwitchIO.xExitBarCylinderRetract:=1;
		  	ConveyorExitIO.xPutInto:=0;
		  	iStep:=4;
		  4:(*下料*)
		  (*通过出料传输线下料*)
		  IF SwitchIO.xExitEnable  AND m_xExitBarDelay AND NOT SwitchIO.xExitBarCylinderRetract  THEN		  
		  	ConveyorExitIO.xUnload:=1;
		  ELSE
		  	ConveyorExitIO.xUnload:=0;
		  END_IF;	
		   (*通过进料传输线下料*)
		  IF SwitchIO.xExitEnable  AND m_xExitBarDelay  AND SwitchIO.xExitBarCylinderRetract THEN		  
		  	ConveyorEntryIO.xUnload:=1;
		  ELSE
		  	ConveyorEntryIO.xUnload:=0;
		  END_IF;			    	
		  IF (ConveyorExitIO.xEmpty OR ConveyorEntryIO.xEmpty) AND m_xExitBarDelay  THEN
		  	ConveyorExitIO.xPutInto:=1;
		  	ConveyorEntryIO.xPutInto:=1;
			iStep:=0; 
		  END_IF;
	END_CASE;
        m_tonLiftCylinderDelay(IN:=NOT ConveyorEntryIO.xEmpty AND iStep=1 ,PT:= T#1S ,Q:= m_xLiftCylinderDelay ,ET:=m_tLiftCylinderDelay );
 		m_tonExitBarDelay(IN:=iStep=4 ,PT:= T#1s ,Q:= m_xExitBarDelay ,ET:= m_tExitBarDelay);
END_IF;
(*复位程序*)
IF g_xReset 
	OR LDP(TRUE,SwitchIO.xLiftCylinderExtendInit) 
	OR LDF(TRUE,SwitchIO.xLiftCylinderExtendInit) 
	OR LDP(TRUE,SwitchIO.xPutInto)  THEN
	ConveyorEntryIO.xPutInto:=1;
	ConveyorExitIO.xPutInto:=1;
	iStep:=0;
END_IF;

IF g_xManual  THEN
	iStep:=0;
	ConveyorEntryIO.xLoad:=0;
    ConveyorEntryIO.xUnload:=0;
	ConveyorEntryIO.xPutInto:=0;
	ConveyorExitIO.xLoad:=0;
	ConveyorExitIo.xUnload:=0;
	ConveyorExitIO.xPutInto:=0;
	SwitchIO.xEntryBarCylinderRetract:=0;
	SwitchIO.xExitBarCylinderRetract:=0;
	IF SwitchIO.xEntryBarCylinderRetractButton THEN
		SwitchIO.xEntryBarCylinderRetract:=1;
	ELSE
		SwitchIO.xEntryBarCylinderRetract:=0;
	END_IF;
		IF SwitchIO.xExitBarCylinderRetractButton THEN
		SwitchIO.xExitBarCylinderRetract:=1;
	ELSE
		SwitchIO.xExitBarCylinderRetract:=0;
		END_IF;
		IF SwitchIO.xLiftCylinderExtendButton AND NOT SwitchIO.xLiftCylinderRetractButton THEN
			SwitchIO.xLiftCylinderExtend:=1;
			SwitchIO.xLiftCylinderRetract:=0;
		END_IF;
		IF NOT SwitchIO.xLiftCylinderExtendButton AND  SwitchIO.xLiftCylinderRetractButton THEN
			SwitchIO.xLiftCylinderExtend:=0;
			SwitchIO.xLiftCylinderRetract:=1;
		END_IF;		 
END_IF;
(*气缸超时报警*)
m_tonCylinderOvertime(IN:= (SwitchIO.xLiftCylinderExtend AND NOT SwitchIO.xLiftCylinderExtendDetect) 
                                                OR  (SwitchIO.xLiftCylinderRetract AND NOT SwitchIO.xLiftCylinderRetractDetect) ,
                                               PT:= SwitchIO.tSetOvertime ,Q:= SwitchIO.xOvertimeAlarm ,ET:= m_tCylinderOvertimeCurrent );
END_FUNCTION_BLOCK
